(* CoDeSys 2.3.9.50 project: 3F.pr6 *)
(* Libraries: STANDARD.LB6 5.6.98 12:03:02 *)

(* POU MAIN, LD *)
PROGRAM MAIN
VAR
	Start AT %IX0.0: BOOL;
	t1: TON;
	Light AT %QX0.0: BOOL;
	t2: TON;
	t3: TON;
	t4: TON;
	t5: TON;
	t6: TON;
	t7: TON;
END_VAR
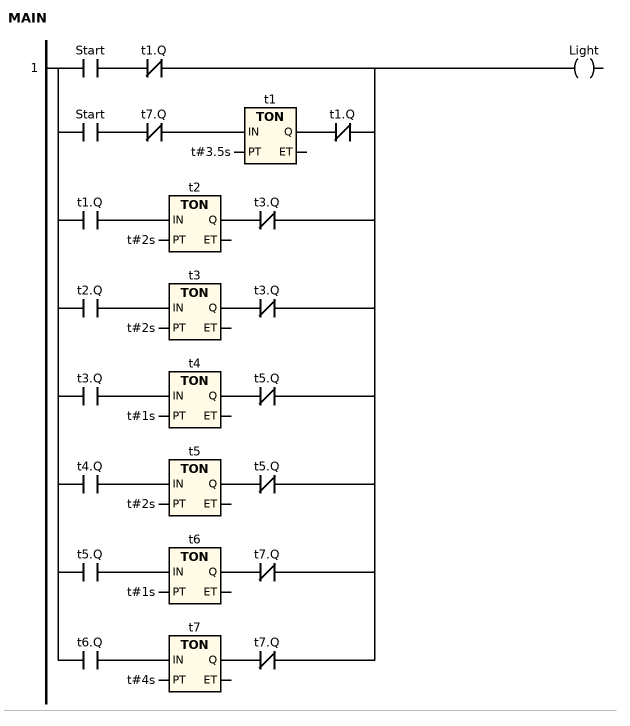
_LD_ (* Ladder Diagram *)
NETWORK 1
	{ [Start] - [/t1.Q] | [Start] - [/t7.Q] - t1:TON(IN: *, PT: t#3.5s) - [/t1.Q] | [t1.Q] - t2:TON(IN: *, PT: t#2s) - [/t3.Q] | [t2.Q] - t3:TON(IN: *, PT: t#2s) - [/t3.Q] | [t3.Q] - t4:TON(IN: *, PT: t#1s) - [/t5.Q] | [t4.Q] - t5:TON(IN: *, PT: t#2s) - [/t5.Q] | [t5.Q] - t6:TON(IN: *, PT: t#1s) - [/t7.Q] | [t6.Q] - t7:TON(IN: *, PT: t#4s) - [/t7.Q] } --- (Light)
_END_LD_
END_PROGRAM
